TYPE STATE:
    STRUCT
        curTime: LREAL;
        dvar_M_aut_x: DINT;
        dvar_M_aut_y: DINT;
        dvar_M_aut_z: DINT;
    END_STRUCT;
END_TYPE
